PROGRAM MAIN
VAR
END_VAR

END_PROGRAM

(* stored: Version 1.1.0.1
   POU MAIN: Id {7ff428b3-db85-4631-8c8c-96d4e1c4c158} *)
